// TIA Portal V18 export
TYPE "UDT_AHUEqp"
// stored: IsFailsafeCompliant false
   STRUCT
      Cfg : "UDT_AHUEqpDataType";
      State { S7_SetPoint := 'True'} : "UDT_AHUEqpDataType";
      Demand { S7_SetPoint := 'True'} : "UDT_AHUEqpDemand";
      LimiterGridOperation { S7_SetPoint := 'True'} : "UDT_AHUsEqpDemandLimiter";
      LimiterDieselOperation { S7_SetPoint := 'True'} : "UDT_AHUsEqpDemandLimiter";
   END_STRUCT;
END_TYPE
